FUNCTION_BLOCK AL_DEMUX_3 (* AL demultiplexor (generic FB) Adapter-Ausgang wird nur bei Wertänderung aktualisiert (Event nur bei tatsächlicher Änderung). *)
  (* Standard: 61499-2; Description: Copyright (c) 2026 HR Agrartechnik GmbH This program and the accompanying materials are made available under the terms of the Eclipse Public License 2.0 which is available at https://www.eclipse.org/legal/epl-2.0/ SPDX-License-Identifier: EPL-2.0 *)
  (* Version 1.0, 2026-05-28, Franz Höpfinger, HR Agrartechnik GmbH *)
  PACKAGE adapter::selection::unidirectional;
  {SET_ATTRIBUTE(eclipse4diac::core::GenericClassName, 'GEN_AL_DEMUX')}
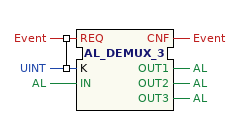
  EVENT_INPUT
    REQ WITH K; (* Set Index K *)
  END_EVENT
  EVENT_OUTPUT
    CNF; (* Confirmation of Set Index K *)
  END_EVENT
  VAR_INPUT
    K : UINT; (* index *)
  END_VAR
  SOCKETS
    IN : adapter::types::unidirectional::AL; (* Input Value to demultiplex *)
  END_SOCKETS
  PLUGS
    OUT1 : adapter::types::unidirectional::AL;
    OUT2 : adapter::types::unidirectional::AL;
    OUT3 : adapter::types::unidirectional::AL;
  END_PLUGS
END_FUNCTION_BLOCK
